// TIA Portal V18 export
TYPE "RCS_PMInterface_V1"
// stored: IsFailsafeCompliant false
   STRUCT
      Enable : Bool;   // Enable Process Module(PM)
      SetInitial : Bool;   // Set PM initial
      InitialRun : Bool;   // PM initial Running
      InitialOK : Bool;   // PM initial completed and OK
      AtHome : Bool;   // PM at home position
      SetNextStep : Bool;   // Set go to next step in StepMode
      GoNextStep : Bool;   // Go to next step in StepMode
      TriggerOneCycle : Bool;   // Trigger PM running One Cycle
      WaitRunning : Bool;   // PM in wait Auto running Status
      Running : Bool;   // PM in Auto running Status
      UnPause : Bool;   // Auto Running Pause (0=Pause)
      ProcessStart : Bool;   // Process start flag
      ProcessComplete : Bool;   // Process complete flag
      Alarm : Bool;   // PM AlarmFlag _Reset-Start
      AlarmImdilyStop : Bool;   // PM Immediately Stop Alram _Reset-Initial
      AlarmCycleStop : Bool;   // PM Cycle Stop Alram
      ProcessStatus : DInt;   // Process running status
      ProcessResult : DInt;   // Process Module Complete product status,0=NA,1=OK,other=NG(101~109)
      OperatorPrompt : UInt;   // PM Operator Prompt
      Num : Int;   // Process Module Number
      StepNum : Int;   // PM flow Step
      SpareByte : Array[0..3] of Byte;
   END_STRUCT;
END_TYPE
